// TIA Portal V20 export
// export: Created 2025-12-01T14:57:44.6955355Z, ExportSetting None, DisplayName Totally Integrated Automation Portal, DisplayVersion V20 Update 3, DisplayName TIA Portal Openness, DisplayVersion V20 Update 3, DisplayName TIA Portal Version Control Interface, DisplayVersion V20 Update 3, DisplayName STEP 7 Professional, DisplayVersion V20 Update 3, DisplayName STEP 7 Safety, DisplayVersion V20 Update 2, DisplayName WinCC Basic/Comfort/Advanced, DisplayVersion V20 Update 3, DisplayName WinCC Professional, DisplayVersion V20 Update 3, DisplayName WinCC Unified, DisplayVersion V20 Update 3
FUNCTION "FC572_Guardar_Datos_Fifo" : Void   // FC572, STL
{ S7_Optimized_Access := 'FALSE' }
// stored: AutoNumber false
   VAR_INPUT
      DB_FIFO_Ordenes : UInt;
      Num_Scanner : UInt;   // Numero de scanner sobre el que se realiza la busqueda
      Long_FIFO : UInt;
      Posicion_FIFO : UInt;
      Datos_Scanner_Cruce : "ROUT_Orden_Fifo_Scanner";
   END_VAR
   VAR_TEMP
      Guardar_AR2 : DWord;
      P_Inicio_Datos : DWord;
      P_Any_Datos : Any;
      NumDB : Word;
      MaxRegistros : UInt;
      LongRegistro : UInt;
      OffsetPrimerRegistro : UInt;
      ValorReturn : Int;
      Elementos_X_Registro : Int;
      Relleno : Byte;
   END_VAR
BEGIN

NETWORK
TITLE = Inicializar Variables
//////////////////////////////////////////////////////////////////////////
/// - Datos del DB a leer

      L     #DB_FIFO_Ordenes;  // - Numero de DB a Leer
      T     #NumDB;
      L     "CTE_MaxMesas";  // - Numero Maximo de Registros
      T     #MaxRegistros;
      L     "ROUT_Long_Reg_Datos_FIFO";  // - Longitud de la estructura del Registro
      T     #LongRegistro;
      L     #Long_FIFO;
      T     #Elementos_X_Registro;
      L     0;  // - Offset del Primer Registro
      T     #OffsetPrimerRegistro;


//////////////////////////////////////////////////////////////////////////


NETWORK
TITLE = Posicionarse en el Registro
//////////////////////////////////////////////////////////////////////////
/// - Comprobar si el registro existe (Maximo de Registros)

      L     #Num_Scanner;
      L     #MaxRegistros;
      >I;
      JC    Error_MaxRegistros;


//////////////////////////////////////////////////////////////////////////
/// - Calculo de la posicion del registro

      L     #Num_Scanner;
      L     #LongRegistro;
      *I;
      L     #Elementos_X_Registro;
      *I;
      L     #OffsetPrimerRegistro;
      +I;
      SLD   3;
      T     #P_Inicio_Datos;


// miramos si tenemos que sacar un registro diferente del primero

      L     #Posicion_FIFO;
      L     1;
      ==I;
      JC    guardar_datos;
// si es un registro diferente del primero, calculamos el offset para colocarnos en el registro correcto

      L     #Posicion_FIFO;
      L     1;
      -I;
      L     #LongRegistro;
      *I;
      SLD   3;
      L     #P_Inicio_Datos;
      +D;
      T     #P_Inicio_Datos;



NETWORK
TITLE = Transferenica del Registro
//////////////////////////////////////////////////////////////////////////
/// - Calculo del Puntero Any de los Datos
guardar_datos:NOP   0;
      TAR2  #Guardar_AR2;  // - Guardar el Puntero AR2

      LAR2  P##P_Any_Datos;  // - Direccion del Puntero Any
      L     B#16#10;  //   10H para S7
      T     LB [AR2, P#0.0];
      L     B#16#2;  //   Tipo de Datos (BYTE)
      T     LB [AR2, P#1.0];
      L     #LongRegistro;  //   Longitud de la Estructura
      T     LW [AR2, P#2.0];
      L     #NumDB;  //   Numero de DB
      T     LW [AR2, P#4.0];
      L     #P_Inicio_Datos;  //   Direccion de Inicio
      T     LD [AR2, P#6.0];
      L     B#16#84;  //   El Area de Memoria = DB
      T     LB [AR2, P#6.0];

      LAR2  #Guardar_AR2;  // - Recuperar el Puntero AR2

//////////////////////////////////////////////////////////////////////////
/// - Transferencia de los Datos a Leer

      CALL  BLKMOV
      ( SRCBLK  := #Datos_Scanner_Cruce,
        RET_VAL := #ValorReturn,
        DSTBLK  := #P_Any_Datos
      );

      L     #ValorReturn;  // - Comprobar que se ha leido el registro
      L     0;
      <>I;
      JC    Error_LecturaDelRegisto;


//////////////////////////////////////////////////////////////////////////
/// - Fin de la Lectura del Registro

      BE;  // - Finalizar bloque



NETWORK
TITLE = Errores en el Sistema de Lectura
//////////////////////////////////////////////////////////////////////////
/// - Numero De Maximo de Registros Sobrepasado

Error_MaxRegistros:NOP   0;
      BE;  // - Finalizar bloque

////////////////////////////////////////////////////
/// - Error a Leer el Registro

Error_LecturaDelRegisto:NOP   0;
      BE;  // - Finalizar bloque


END_FUNCTION
